PROGRAM MAIN
VAR
	PLCVar AT %MD0 : DWORD;
	PCVar AT %MD1 : DWORD;
	TP_1		: TP;
	TOGGEL: BOOL;
END_VAR

TOGGEL := NOT TOGGEL;
TP_1( IN := TOGGEL, PT := T#4S);
IF (TP_1.Q = 0) THEN
	PLCVar := PLCVar + 1;
	TOGGEL := NOT TOGGEL;
	TP_1( IN := TOGGEL, PT := T#4S);
END_IF

END_PROGRAM

(* stored: Version 1.1.0.1, ProductVersion 3.1.4024.5
   POU MAIN: Id {5b1611da-9a64-4e17-938b-8f9045a51963}, SpecialFunc None *)
